Staubli VAL3: getListSession.pgx

public program getListSession(string& x_sSession[] (dimensions=1))
begin
  // Build the list
  libList("session",x_sSession)
end
